Universal Robots PolyScope program: Lab_exe_9_2_154.urp

Program Lab_exe_9_2_154 (createdIn=3.2.19293 lastSavedIn=3.2.19293 directory=/programs installation=default robotSerialNumber=2015351391)
Calibrated DH parameters: a=[0.000352, -0.161198, -0.373486, 0.00005, 0.000049, 0]; d=[0.089268, 352.477598, -320.08558, -32.281492, 0.094939, 0.082518]; alpha=[1.570728, 0.001116, -0.003686, 1.571189, -1.570572, 0]; deltaTheta=[-0.000012, 1.181849, -1.491165, 0.309495, -0.000007, 0.000025]
Robot Program (runOnlyOnce=false motionType=MoveJ speed=1.047198 acceleration=1.396263 recalculateMotions=false)
  Wait Sleep waitTime=0.01
  If MODBUS_3≟ True
    Set ExpressionOutput pin=MODBUS_1; expression=True
    Popup Message (haltProgram=false message=modbus output is True)
  If MODBUS_4≟ True
    Set ExpressionOutput pin=MODBUS_2; expression=True
    Popup Message (haltProgram=false message=modbus output is True)
Thread 线程_1 (runOnlyOnce=false trackProgramExecution=false)
  Wait Sleep waitTime=0.01
  If MODBUS_3≟ True
    Wait Sleep waitTime=5
    If MODBUS_1≟ False
      Popup Message (haltProgram=false message=no modbus output.)
  If MODBUS_4≟ True
    Wait Sleep waitTime=5
    If MODBUS_2≟ False
      Popup Message (haltProgram=false message=no modbus output.)
